// TIA Portal V16 export
// export: Created 2023-03-29T11:05:02.5391447Z, ExportSetting WithDefaults, DisplayName Totally Integrated Automation Portal, DisplayVersion V16 Update 6, DisplayName TIA Portal Version Control Interface, DisplayVersion V16 Update 2, DisplayName TIA Portal Openness, DisplayVersion V16 Update 6, DisplayName STEP 7 Professional, DisplayVersion V16 Update 6, DisplayName STEP 7 Safety, DisplayVersion V16, DisplayName WinCC Advanced, DisplayVersion V16 Update 6
DATA_BLOCK "dbTimersForDrivers"   // DB4
{ S7_Optimized_Access := 'FALSE' }
VERSION : 0.1
// stored: AutoNumber true, DBAccessibleFromOPCUA true, IsOnlyStoredInLoadMemory false, IsWriteProtectedInAS false
   VAR
      TimerP1 { S7_SetPoint := 'True'} : IEC_TIMER;   // Timer drivera
      TimerP2 { S7_SetPoint := 'True'} : IEC_TIMER;   // Timer drivera
      TimerP3 { S7_SetPoint := 'True'} : IEC_TIMER;   // Timer drivera
      ResetModeAut { S7_SetPoint := 'True'} : IEC_TIMER;   // Delay Reset Mode Work Aut
      TimerZ11 { S7_SetPoint := 'True'} : IEC_TIMER;   // Timer drivera Z11
      TimerZ12 { S7_SetPoint := 'True'} : IEC_TIMER;   // Timer drivera Z12
      TimerP4 { S7_SetPoint := 'True'} : IEC_TIMER;   // Timer drivera
      Timer_OFF_Inverter_P1 { S7_SetPoint := 'True'} : IEC_TIMER;   // Timer blokowania dołączenie stycznika falownika P1
      Timer_OFF_Inverter_P2 { S7_SetPoint := 'True'} : IEC_TIMER;   // Timer blokowania dołączenie stycznika falownik P2
      Timer_OFF_Inverter_P3 { S7_SetPoint := 'True'} : IEC_TIMER;   // Timer blokowania dołączenie stycznika falownik P3
      Timer_OFF_Inverter_P4 { S7_SetPoint := 'True'} : IEC_TIMER;   // Timer blokowania dołączenie stycznika falownik P4
      Timer_Start_Network_P1 { S7_SetPoint := 'True'} : IEC_TIMER;   // Timer opóźnienia przełaczenia na sieć
      Timer_Start_Network_P2 { S7_SetPoint := 'True'} : IEC_TIMER;   // Timer opóźnienia przełaczenia na sieć
      Timer_Start_Network_P3 { S7_SetPoint := 'True'} : IEC_TIMER;   // Timer opóźnienia przełaczenia na sieć
      Timer_Start_Network_P4 { S7_SetPoint := 'True'} : IEC_TIMER;   // Timer opóźnienia przełaczenia na sieć
      Timer_Start_Inver_P1 { S7_SetPoint := 'True'} : IEC_TIMER;   // Timer opóźnienia przełaczenia na falownik
      Timer_Start_Inver_P2 { S7_SetPoint := 'True'} : IEC_TIMER;   // Timer opóźnienia przełaczenia na falownik
      Timer_Start_Inver_P3 { S7_SetPoint := 'True'} : IEC_TIMER;   // Timer opóźnienia przełaczenia na falownik
      Timer_Start_Inver_P4 { S7_SetPoint := 'True'} : IEC_TIMER;   // Timer opóźnienia przełaczenia na falownik
      Timer_Hiteresis_On_Set50Hz_Inver_P1 { S7_SetPoint := 'True'} : IEC_TIMER;   // Timer opóźnieniawyłączeniea falownika
      Timer_Hiteresis_On_Set50Hz_Inver_P2 { S7_SetPoint := 'True'} : IEC_TIMER;   // Timer opóźnieniawyłączeniea falownika
      Timer_Hiteresis_On_Set50Hz_Inver_P3 { S7_SetPoint := 'True'} : IEC_TIMER;   // Timer opóźnieniawyłączeniea falownika
      Timer_Hiteresis_On_Set50Hz_Inver_P4 { S7_SetPoint := 'True'} : IEC_TIMER;   // Timer opóźnieniawyłączeniea falownika
      ResetBit_KasowaniaAlarm { S7_SetPoint := 'True'} : IEC_TIMER;   // Timer impulsu kasowania bitu kasowania alarmów HMI
      TimerAlarm_1 { S7_SetPoint := 'True'} : IEC_TIMER;   // Timer impulsu kasowania bitu kasowania alarmów HMI
   END_VAR
BEGIN
   TimerP1.PT := T#10S;
   TimerP2.PT := T#10S;
   TimerP3.PT := T#10S;
   ResetModeAut.PT := T#2S;
   TimerZ11.PT := T#30S;
   TimerZ12.PT := T#30S;
   TimerP4.PT := T#10S;
   Timer_OFF_Inverter_P1.PT := T#5S;
   Timer_OFF_Inverter_P2.PT := T#5S;
   Timer_OFF_Inverter_P3.PT := T#5S;
   Timer_OFF_Inverter_P4.PT := T#5S;
   Timer_Start_Network_P1.PT := T#3S;
   Timer_Start_Network_P2.PT := T#3S;
   Timer_Start_Network_P3.PT := T#3S;
   Timer_Start_Network_P4.PT := T#3S;
   Timer_Start_Inver_P1.PT := T#3100ms;
   Timer_Start_Inver_P2.PT := T#3200ms;
   Timer_Start_Inver_P3.PT := T#3300ms;
   Timer_Start_Inver_P4.PT := T#3400ms;
   Timer_Hiteresis_On_Set50Hz_Inver_P1.PT := T#10ms;
   Timer_Hiteresis_On_Set50Hz_Inver_P2.PT := T#10ms;
   Timer_Hiteresis_On_Set50Hz_Inver_P3.PT := T#10ms;
   Timer_Hiteresis_On_Set50Hz_Inver_P4.PT := T#10ms;
   ResetBit_KasowaniaAlarm.PT := T#2S;
   TimerAlarm_1.PT := T#5M;
END_DATA_BLOCK
